{attribute 'linkalways'} 
{attribute 'no_explicit_call' := 'This FB is a CLASS and must be accessed using methods or properties'}
{attribute 'enable_dynamic_creation'}
FUNCTION_BLOCK Node_ContainerType_Vector_TcVnVector4_USINT EXTENDS Node
VAR
    out : _GUID;
END_VAR

METHOD PUBLIC  Clone : I_Node
VAR
	pNode : POINTER TO Node_ContainerType_Vector_TcVnVector4_USINT;
END_VAR
pNode := __NEW(Node_ContainerType_Vector_TcVnVector4_USINT);
Clone := pNode^;
END_METHOD

METHOD FB_init : BOOL
VAR_INPUT
	bInitRetains : BOOL; // if TRUE, the retain variables are initialized (warm start / cold start)
	bInCopyCode : BOOL;  // if TRUE, the instance afterwards gets moved into the copy code (online change)
END_VAR
AddOutput('out', out);
END_METHOD

METHOD PROTECTED OnExecute
out.Value := ContainerType_Vector_TcVnVector4_USINT;
END_METHOD

END_FUNCTION_BLOCK

(* stored: Version 1.1.0.1, ProductVersion 3.1.4026.17
   POU Node_ContainerType_Vector_TcVnVector4_USINT: Id {acdebec7-cca3-01f9-0c0e-9562fa345af5}, SpecialFunc None
   Folder Constructor: Id {536ba967-3fd4-007c-2d5c-91258bb130fa}
   Method Clone: Id {993d8bd1-8b7f-06ab-1679-bae0509feff8}
   Method FB_init: Id {13d05073-beb0-0c17-045e-58816fcfd743}
   Method OnExecute: Id {db6eae20-8c0c-010f-3359-f3b3258c1d82} *)
